FUNCTION_BLOCK FB_Puls
VAR_INPUT
	tPeriod  :TIME;
END_VAR
VAR_OUTPUT
	bPuls 	 :BOOL;
END_VAR
VAR
	bM1		 :BOOL := TRUE;
	TP1		 :TP;
	TP2		 :TP;
	fbPulsM1 :F_TRIG;
	iCounter :INT;
	bM2		 :BOOL;
	fbPulsM2 :F_TRIG;
END_VAR

fbPulsM1(CLK:= bM1);
TP1(IN:= fbPulsM1.Q, PT:=tPeriod);
bM2 :=TP1.Q;

fbPulsM2(CLK:= bM2);
TP2(IN:= fbPulsM1.Q,  PT:=tPeriod);

bM1:= TP2.Q;
bPuls := bM1;
IF fbPulsM1.Q THEN
	iCounter:=iCounter+1;
END_IF

END_FUNCTION_BLOCK

(* stored: Version 1.1.0.1, ProductVersion 3.1.4024.4
   POU FB_Puls: Id {03cc3659-2869-4289-acd0-a091a4802cb0}, SpecialFunc None *)
